// Mitsubishi GX Works2 project: ZhaoQing_HuaCheng1_12_15_8_55   PLC: Q03UDE

TYPE ConveyorIO : STRUCT
  xCWPresent : BOOL;  (* 正转检测有无传感器 *)
  xCCWPresent : BOOL;  (* 反转检测有无传感器 *)
  xLoad : BOOL;  (* 上料请求 *)
  xUnload : BOOL;  (* 下料请求 *)
  xMotorCW : BOOL;  (* 电机正转 *)
  xMotorCCW : BOOL;  (* 电机反转 *)
  xEmpty : BOOL;  (* 线体状态为空 *)
  xNextRun : BOOL;  (* 下段线体运行 *)
  xUnloadCCW : BOOL;  (* 下料为反转 *)
  xloadCCW : BOOL;  (* 上料为反转 *)
  xForward : BOOL;  (* 正转手动 *)
  xBackward : BOOL;  (* 反转手动 *)
  xBusy : BOOL;  (* 工作中 *)
  xPutInto : BOOL;  (* 线体直接投入物料 *)
  xLoadAlarrm : BOOL;  (* 上料报警 *)
  xUnloadAlarm : BOOL;  (* 下料报警 *)
  iProductCategory : INT;  (* 产品种类 *)
  tLoadDelay : TIME;  (* 进入延时设置 *)
  tUnloadAlarmDelay : TIME;  (* 下料时间设置 *)
  xNotArriveAlarm : BOOL;  (* 未到达报警 *)
END_STRUCT END_TYPE

TYPE ShuttleCarIO : STRUCT
  xReady : BOOL;  (* 准备就绪 *)
  xForward : BOOL;  (* 正转 *)
  xBackward : BOOL;  (* 反转 *)
  iCurrentPos : INT;  (* 当前位置 *)
  iDestinationPos : INT;  (* 目标位置 *)
  xCW : BOOL;  (* 正转输出 *)
  xCCW : BOOL;  (* 反转输出 *)
  xBrake : BOOL;  (* 刹车 *)
  xHomeSwitch : BOOL;  (* 零位接近开关 *)
  xPosLimit : BOOL;  (* 正限位 *)
  xNegLimit : BOOL;  (* 负限位 *)
  xMDIExe : BOOL;  (* MDI开始 *)
  xMDIDone : BOOL;  (* MDI 完成 *)
  xPassLimit : BOOL;  (* 限位屏蔽 *)
  xPosLimitCatch : BOOL;  (* 正限位捕捉 *)
  xNegLimitCatch : BOOL;  (* 负限位捕捉 *)
  xHomeExe : BOOL;  (* 开始寻零 *)
  xHomeDone : BOOL;  (* 寻零完成 *)
  xHomeBusy : BOOL;  (* 寻零中 *)
  xHomeFailed : BOOL;  (* 寻零失败 *)
  xBusy : BOOL;  (* 工作中 *)
END_STRUCT END_TYPE

TYPE SwitchIO : STRUCT
  xLiftCylinderRetractDetect : BOOL;
  xLiftCylinderExtendDetect : BOOL;
  xLiftCylinderRetract : BOOL;
  xLiftCylinderExtend : BOOL;
  xEntryBarCylinderRetract : BOOL;
  xLiftCylinderExtendInit : BOOL;
  xEntryEnable : BOOL;
  xExitEnable : BOOL;
  xExitBarCylinderRetract : BOOL;
  xSwithEnable : BOOL;
  xLiftCylinderRetractButton : BOOL;
  xLiftCylinderExtendButton : BOOL;
  xEntryBarCylinderRetractButton : BOOL;
  xExitBarCylinderRetractButton : BOOL;
END_STRUCT END_TYPE

// global labels: Global1
VAR_GLOBAL
  g_xAuto : BOOL;
  g_xManual : BOOL;
  g_xEStop AT X23 : BOOL;
  g_xReset AT X20 : BOOL;
  g_xStackLampRed AT Y120 : BOOL;
  g_xStackLampAmber AT Y121 : BOOL;
  g_xStackLampGreen AT Y122 : BOOL;
  g_xBuzzer AT Y123 : BOOL;
  g_xStop AT M2 : BOOL;
  g_xLocalAutoStart AT M1 : BOOL;
  g_xRemoteAutoStart AT M0 : BOOL;
  g_xRemoteAuto AT M10 : BOOL;
  g_iState AT D40 : INT;
  g_iLocalAutoStep : INT;
  g_xAlarm : BOOL;
END_VAR

// task Task_01 (event TRUE, interval 0, priority 31): POU, Start, UDP

PROGRAM POU
VAR
  H3000Conveyor1 : Conveyor;
  H3000Conveyor1IO : ConveyorIO;
  H3000Conveyor2 : Conveyor;
  H3000Conveyor2IO : ConveyorIO;
  H3000Conveyor3 : Conveyor;
  H3000Conveyor3IO : ConveyorIO;
  H3000Conveyor4 : Conveyor;
  H3000Conveyor4IO : ConveyorIO;
  H3000Conveyor5 : Conveyor;
  H3000Conveyor5IO : ConveyorIO;
  H3000Conveyor6 : Conveyor;
  H3000Conveyor6IO : ConveyorIO;
  H3000Conveyor7 : Conveyor;
  H3000Conveyor7IO : ConveyorIO;
  H3000Conveyor8 : Conveyor;
  H3000Conveyor8IO : ConveyorIO;
  H3000Conveyor9 : Conveyor;
  H3000Conveyor9IO : ConveyorIO;
  H3000Conveyor10 : Conveyor;
  H3000Conveyor10IO : ConveyorIO;
  H3000ChemConveyor1 : Conveyor;
  H3000ChemConveyor1IO : ConveyorIO;
  H3000ChemConveyor2 : Conveyor;
  H3000ChemConveyor2IO : ConveyorIO;
  H3000ChemConveyor3 : Conveyor;
  H3000ChemConveyor3IO : ConveyorIO;
  Lifter1 : ShuttleCar;
  Lifter1IO : ShuttleCarIO;
  Conveyor1 : Conveyor;
  Conveyor1IO : ConveyorIO;
  Lifter2 : ShuttleCar;
  Lifter2IO : ShuttleCarIO;
  Conveyor2 : Conveyor;
  Conveyor2IO : ConveyorIO;
  H2200Conveyor1 : Conveyor;
  H2200Conveyor1IO : ConveyorIO;
  H2200Conveyor2 : Conveyor;
  H2200Conveyor2IO : ConveyorIO;
  H2200Conveyor3 : Conveyor;
  H2200Conveyor3IO : ConveyorIO;
  H2200Conveyor4 : Conveyor;
  H2200Conveyor4IO : ConveyorIO;
  H2200Conveyor5 : Conveyor;
  H2200Conveyor5IO : ConveyorIO;
  H2200Conveyor6 : Conveyor;
  H2200Conveyor6IO : ConveyorIO;
  H2200Conveyor7 : Conveyor;
  H2200Conveyor7IO : ConveyorIO;
  H2200Conveyor8 : Conveyor;
  H2200Conveyor8IO : ConveyorIO;
  H2200Conveyor9 : Conveyor;
  H2200Conveyor9IO : ConveyorIO;
  H2200Conveyor10 : Conveyor;
  H2200Conveyor10IO : ConveyorIO;
  H1000Conveyor1 : Conveyor;
  H1000Conveyor1IO : ConveyorIO;
  H1000Conveyor2 : Conveyor;
  H1000Conveyor2IO : ConveyorIO;
  H1000Conveyor3 : Conveyor;
  H1000Conveyor3IO : ConveyorIO;
  H1000Conveyor4 : Conveyor;
  H1000Conveyor4IO : ConveyorIO;
  H1000Conveyor5 : Conveyor;
  H1000Conveyor5IO : ConveyorIO;
  H1000Conveyor6 : Conveyor;
  H1000Conveyor6IO : ConveyorIO;
  H1000Conveyor7 : Conveyor;
  H1000Conveyor7IO : ConveyorIO;
  H1000Conveyor8 : Conveyor;
  H1000Conveyor8IO : ConveyorIO;
  H1000Conveyor9 : Conveyor;
  H1000Conveyor9IO : ConveyorIO;
  H3000SwitchChem : Switch;
  H3000SwitchChemIO : SwitchIO;
  H850Switch : Switch;
  H850SwitchIO : SwitchIO;
  H850SwitchConveyorIn : ConveyorIO;
  H850SwitchConveyorOut : ConveyorIO;
  H850Conveyor8 : Conveyor;
  H850Conveyor8IO : ConveyorIO;
  H1000Conveyor10 : Conveyor;
  H1000Conveyor10IO : ConveyorIO;
  H3000SwitchChemConveyorIn : ConveyorIO;
  H3000SwitchChemConveyorOut : ConveyorIO;
  H3000SwitchQuadPackage : Switch;
  H3000SwitchQuadPackageIO : SwitchIO;
  H3000SwitchPackageConveyorIn : ConveyorIO;
  H3000SwitchPackageConveyorOut : ConveyorIO;
  H2200Switch1 : Switch;
  H2200Switch1IO : SwitchIO;
  H2200Switch1ConveyorIn : ConveyorIO;
  H2200Switch1ConveyorOut : ConveyorIO;
  H2200Switch2 : Switch;
  H2200Switch2IO : SwitchIO;
  H2200Switch2ConveyorIn : ConveyorIO;
  H2200Switch2ConveyorOut : ConveyorIO;
  iStep : INT;
  Import1Conveyor1 : Conveyor;
  Import1Conveyor1IO : ConveyorIO;
  Import1Conveyor2 : Conveyor;
  Import1Conveyor2IO : ConveyorIO;
  Import2Conveyor1 : Conveyor;
  Import2Conveyor1IO : ConveyorIO;
  Import2Conveyor2 : Conveyor;
  Import2Conveyor2IO : ConveyorIO;
  Export1Conveyor1 : Conveyor;
  Export1Conveyor1IO : ConveyorIO;
  Export1Conveyor2 : Conveyor;
  Export1Conveyor2IO : ConveyorIO;
  Export2Conveyor1 : Conveyor;
  Export2Conveyor1IO : ConveyorIO;
  Export2Conveyor2 : Conveyor;
  Export2Conveyor2IO : ConveyorIO;
  Export2Switch : Switch;
  Export2SwitchIO : SwitchIO;
  Export2SwitchConveyorIn : ConveyorIO;
  Export2SwitchConveyorOut : ConveyorIO;
  H850Rotor : ShuttleCar;
  H850RotorIO : ShuttleCarIO;
  H850RotorConveyor : Conveyor;
  H850RotorConveyorIO : ConveyorIO;
  H2200RotorIO : ShuttleCarIO;
  H2200RotorConveyor : Conveyor;
  H2200RotorConveyorIO : ConveyorIO;
  H2200Rotor : ShuttleCar;
  H850Conveyor1 : Conveyor;
  H850Conveyor1IO : ConveyorIO;
  H850Conveyor3 : Conveyor;
  H850Conveyor3IO : ConveyorIO;
  H850Conveyor4 : Conveyor;
  H850Conveyor4IO : ConveyorIO;
  H850Conveyor5 : Conveyor;
  H850Conveyor5IO : ConveyorIO;
  H850Conveyor6 : Conveyor;
  H850Conveyor6IO : ConveyorIO;
  Lifter2Position : ARRAY [0..5] OF INT;
  ii : INT;  (* 提升机2任务号 *)
  H2200SwitchEmptyABack : Switch;
  H2200SwitchEmptyABackIO : SwitchIO;
  H2200SwitchEmptyABackConveyorIn : ConveyorIO;
  H2200SwitchEmptyABackConveyorOut : ConveyorIO;
  H2200SwitchEmptyBBack : Switch;
  H2200SwitchEmptyBBackIO : SwitchIO;
  H2200SwitchEmptyBBackConveyorIn : ConveyorIO;
  H2200SwitchEmptyBBackConveyorOut : ConveyorIO;
  H2200ImportConveyor1 : Conveyor;
  H2200ImportConveyor1IO : ConveyorIO;
  H2200ImportConveyor2 : Conveyor;
  H2200ImportConveyor2IO : ConveyorIO;
  Import1Switch : Switch;
  Import1SwitchIO : SwitchIO;
  Import1SwitchConveyorIn : ConveyorIO;
  Import1SwitchConveyorOut : ConveyorIO;
  Export1Switch : Switch;
  Export1SwitchIO : SwitchIO;
  Export1SwitchConveyorIn : ConveyorIO;
  Export1SwitchConveyorOut : ConveyorIO;
  Import2Switch : Switch;
  Import2SwitchIO : SwitchIO;
  Import2SwitchConveyorIn : ConveyorIO;
  Import2SwitchConveyorOut : ConveyorIO;
  Import1LoadCylinder : ShuttleCar;
  Import1LoadCylinderIO : ShuttleCarIO;
  Import2LoadCylinder : ShuttleCar;
  Import2LoadCylinderIO : ShuttleCarIO;
  Export1LoadCylinder : ShuttleCar;
  Export1LoadCylinderIO : ShuttleCarIO;
  Export2LoadCylinder : ShuttleCar;
  Export2LoadCylinderIO : ShuttleCarIO;
  Lifter2ExportChem : BOOL;  (* 提升机2满框去化成 *)
  Lifter2TaskID : INT;  (* 提升机2动作步骤 *)
  Lifter2Task : PriorityFB;
  H2200Switch1Task : PriorityFB;
  H2200Switch1TaskID : INT;
  H2200Switch1EmptyImport : BOOL;  (* 空框返回入库 *)
  Lifter1Speed : ShuttleCarVelocityFB;
END_VAR
H3000SwitchQuadPackage(ConveyorEntryIO:=H3000SwitchPackageConveyorIn ,
                                                        ConveyorExitIO:=H3000SwitchPackageConveyorOut ,
                                                        SwitchIO:=H3000SwitchQuadPackageIO );
H3000SwitchQuadPackageIO.xLiftCylinderExtendButton:=M75;
H3000SwitchQuadPackageIO.xLiftCylinderRetractButton:=M76;
H3000SwitchQuadPackageIO.xExitBarCylinderRetractButton:=M83;
Y128:=H3000SwitchQuadPackageIO.xEXITBarCylinderRetract;
Y12C:=H3000SwitchQuadPackageIO.xLiftCylinderExtend;
Y12A:=H3000SwitchQuadPackageIO.xLiftCylinderRetract;
H3000SwitchQuadPackageIO.xLiftCylinderExtendDetect:=X29;
H3000SwitchQuadPackageIO.xLiftCylinderRetractDetect:=X2A;
H3000SwitchPackageConveyorIn.xForward:=M77;
H3000SwitchPackageConveyorIn.xCWPresent:=X28;
(*Y187:=H3000SwitchPackageConveyorIn.xMotorCW;*)
H3000SwitchPackageConveyorOut.xForward:=M78;
H3000SwitchPackageConveyorOut.xCWPresent:=X2B;
Y12B:=H3000SwitchPackageConveyorOut.xMotorCW;

H3000SwitchChem(ConveyorEntryIO:=H3000SwitchChemConveyorIn ,
                                                        ConveyorExitIO:=H3000SwitchChemConveyorOut ,
                                                        SwitchIO:=H3000SwitchChemIO );
H3000SwitchChemIO.xLiftCylinderExtendButton:=M79;
H3000SwitchChemIO.xLiftCylinderRetractButton:=M80;
Y129:=H3000SwitchChemIO.xLiftCylinderExtend;
Y12D:=H3000SwitchChemIO.xLiftCylinderRetract;
H3000SwitchChemIO.xLiftCylinderExtendDetect:=X2C;
H3000SwitchChemIO.xLiftCylinderRetractDetect:=X2D;
H3000SwitchChemConveyorIn.xForward:=M81;
H3000SwitchChemConveyorIn.xCWPresent:=X27;
(*Y19B:=H3000SwitchPackageConveyorIn.xMotorCW;*)
H3000SwitchChemConveyorOut.xForward:=M82;
H3000SwitchChemConveyorOut.xCWPresent:=X2E;
Y12E:=H3000SwitchChemConveyorOut.xMotorCW;
H3000SwitchChemIO.xSwithEnable:=1;

Lifter1(ShuttleCarInOut:=Lifter1IO);
ShuttleCarCurrentPosition(X8C OR X8D ,X8C ,X8D, FALSE, Lifter1IO.iCurrentPos);
Lifter1Speed(xEnable:= g_xAuto,
                        xMotorCW:= Lifter1IO.xCW ,
                        xMotorCCW:= Lifter1IO.xCCW,
                        xPosition1Switch:= X8C,
                        xDecelerationSwitch:= X8B ,
	                    xPosition2Switch:= X8D ,
	                    xHighSpeed:= Y18F );
Lifter1IO.xReady:=X24;
Lifter1Io.xForward:=M50 OR X91;
Lifter1IO.xBackward:=M51 OR X92;
Lifter1IO.xPosLimit:=X8E;
Lifter1IO.xNegLimit:=X8F;
Y18D:=Lifter1IO.xCW;
Y18E:=Lifter1IO.xCCW;
Y192:=Lifter1IO.xBrake;

Conveyor1(ConveyorMotor:=Conveyor1IO);
Conveyor1IO.xForward:=M52;
Conveyor1IO.xBackward:=M53;
Conveyor1IO.xCWPresent:=X93;
Conveyor1IO.xCCWPresent:=X94;
Y18B:=Conveyor1IO.xMotorCW;
Y18C:=Conveyor1IO.xMotorCCW;
(*2号提升机*)
Lifter2(ShuttleCarInOut:=Lifter2IO);
Lifter2Position[0]:=0;
Lifter2Position[1]:=57;
Lifter2Position[2]:=590;
Lifter2Position[3]:=5828;
Lifter2Position[4]:=6202;
Lifter2Position[5]:=9200;
Y195:=ShuttleCarVelocityEncoder( g_xAuto , D190 , Lifter2Position[Lifter2IO.iDestinationPos] );
IF LDP(TRUE,g_xAuto) THEN
	Lifter2IO.iCurrentPos:=0;
END_IF;
FOR ii:=0 TO 5 BY 1 DO
	IF abs(D190-Lifter2Position[ii])<5 THEN
		Lifter2IO.iCurrentPos:=ii;
	END_IF;
END_FOR;
Lifter2IO.xReady:=X25;
(*提升机占用标志位控制*)
Lifter2Task(xCondition1:= NOT H850Conveyor8IO.xEmpty ,
                     xCondition2:= NOT H1000Conveyor1IO.xEmpty ,
                     xCondition3:= NOT H3000ChemConveyor3IO.xEmpty  AND Lifter2ExportChem ,
                     xCondition4:= NOT H3000ChemConveyor3IO.xEmpty  AND NOT Lifter2ExportChem ,
                     xCondition5:= FALSE ,
	                 xTaskComplete:= (Lifter2IO.iCurrentPos=3 OR Lifter2IO.iCurrentPos=4) AND LDP(TRUE,Conveyor2IO.xEmpty)  ,
	                 xReset:= g_xReset,
	                 iPriority:=  Lifter2TaskID );
Lifter2Io.xForward:=M54 OR X9B;
Lifter2IO.xBackward:=M55 OR X9C;
Lifter2IO.xPosLimit:=X98;
Lifter2IO.xNegLimit:=X99;
Y193:=Lifter2IO.xCW;
Y194:=Lifter2IO.xCCW;
Y198:=Lifter2IO.xBrake;
(*提升机2编码器清零，到达负限位后清零*)
IF NOT Lifter2IO.xNegLimit THEN
	Y125:=1;
ELSE
	Y125:=0;
END_IF;

Conveyor2(ConveyorMotor:=Conveyor2IO);
Conveyor2IO.xForward:=M56;
Conveyor2IO.xBackward:=M57;
Conveyor2IO.xCWPresent:=X9D;
Conveyor2IO.xCCWPresent:=X9E;
Y19A:=Conveyor2IO.xMotorCW;
Y199:=Conveyor2IO.xMotorCCW;

(*去二封线体*)
H3000Conveyor1(ConveyorMotor:=H3000Conveyor1IO);
H3000Conveyor1IO.xForward:=M30;
H3000Conveyor1IO.xCWPresent:=X2F;
Y12F:=H3000Conveyor1IO.xMotorCW;

H3000Conveyor2(ConveyorMotor:=H3000Conveyor2IO);
H3000Conveyor2IO.xForward:=M31;
H3000Conveyor2IO.xCWPresent:=X30;
Y130:=H3000Conveyor2IO.xMotorCW;

H3000Conveyor3(ConveyorMotor:=H3000Conveyor3IO);
H3000Conveyor3IO.xForward:=M32;
H3000Conveyor3IO.xCWPresent:=X31;
Y131:=H3000Conveyor3IO.xMotorCW;

H3000Conveyor4(ConveyorMotor:=H3000Conveyor4IO);
H3000Conveyor4IO.xForward:=M33;
H3000Conveyor4IO.xCWPresent:=X32;
Y132:=H3000Conveyor4IO.xMotorCW;

H3000Conveyor5(ConveyorMotor:=H3000Conveyor5IO);
H3000Conveyor5IO.xForward:=M34;
H3000Conveyor5IO.xCWPresent:=X33;
Y133:=H3000Conveyor5IO.xMotorCW;

H3000Conveyor6(ConveyorMotor:=H3000Conveyor6IO);
H3000Conveyor6IO.xForward:=M34;
H3000Conveyor6IO.xCWPresent:=X34;
Y134:=H3000Conveyor6IO.xMotorCW;

H3000Conveyor7(ConveyorMotor:=H3000Conveyor7IO);
H3000Conveyor7IO.xForward:=M35;
H3000Conveyor7IO.xCWPresent:=X35;
Y135:=H3000Conveyor7IO.xMotorCW;
H3000Conveyor8(ConveyorMotor:=H3000Conveyor8IO);
H3000Conveyor8IO.xForward:=M36;
H3000Conveyor8IO.xCWPresent:=X36;
Y136:=H3000Conveyor8IO.xMotorCW;

H3000Conveyor9(ConveyorMotor:=H3000Conveyor9IO);
H3000Conveyor9IO.xForward:=M37;
H3000Conveyor9IO.xCWPresent:=X37;
Y137:=H3000Conveyor9IO.xMotorCW;

H3000Conveyor10(ConveyorMotor:=H3000Conveyor10IO);
H3000Conveyor10IO.xForward:=M38;
H3000Conveyor10IO.xCWPresent:=X38;
Y138:=H3000Conveyor10IO.xMotorCW;

(*本段线体没有接线*)
(*H3000ChemConveyor1(ConveyorMotor:=H3000ChemConveyor1IO);
H3000ChemConveyor1IO.xForward:=M39;
H3000ChemConveyor1IO.xCWPresent:=X39;
Y139:=H3000ChemConveyor1IO.xMotorCW;*)

(*去化成H3000线体*)
H3000ChemConveyor2(ConveyorMotor:=H3000ChemConveyor2IO);
H3000ChemConveyor2IO.xForward:=M40;
H3000ChemConveyor2IO.xCWPresent:=X39;
Y13A:=H3000ChemConveyor2IO.xMotorCW;

H3000ChemConveyor3(ConveyorMotor:=H3000ChemConveyor3IO);
H3000ChemConveyor3IO.xForward:=M41;
H3000ChemConveyor3IO.xCWPresent:=X3B;
Y13B:=H3000ChemConveyor3IO.xMotorCW;
(*入库线体*)
H2200Switch1(ConveyorEntryIO:=H2200Switch1ConveyorIn ,
                                                        ConveyorExitIO:=H2200Switch1ConveyorOut ,
                                                        SwitchIO:=H2200Switch1IO );
H2200Switch1Task(xCondition1:=NOT  H2200SwitchEmptyABackConveyorIn.xEmpty AND H2200Switch1EmptyImport,
                                    xCondition2:= NOT  H2200SwitchEmptyBBackConveyorIn.xEmpty AND H2200Switch1EmptyImport,
                                    xCondition3:=NOT  H2200SwitchEmptyABackConveyorIn.xEmpty AND NOT H2200Switch1EmptyImport  ,
                                    xCondition4:=(* NOT  H2200SwitchEmptyBBackConveyorIn.xEmpty AND NOT H2200Switch1EmptyImport*)FALSE,
                                    xCondition5:= NOT H2200ImportConveyor2IO.xEmpty  ,
	                               xTaskComplete:= LDP(TRUE, H2200Switch1ConveyorIn.xEmpty) OR LDP(TRUE, H2200Switch1ConveyorOut.xEmpty)  ,
	                               xReset:= g_xReset ,
	                               iPriority:= H2200Switch1TaskID);
H2200Switch1IO.xLiftCylinderExtendButton:=M84;
H2200Switch1IO.xLiftCylinderRetractButton:=M85;
H2200Switch1IO.xExitBarCylinderRetractButton:=M86;
Y158:=H2200Switch1IO.xEXITBarCylinderRetract;
Y155:=H2200Switch1IO.xLiftCylinderExtend;
Y156:=H2200Switch1IO.xLiftCylinderRetract;
H2200Switch1IO.xLiftCylinderExtendDetect:=X55;
H2200Switch1IO.xLiftCylinderRetractDetect:=X56;
H2200Switch1ConveyorIn.xForward:=M87;
H2200Switch1ConveyorIn.xCWPresent:=X57;
(*Y177:=H2200Switch1ConveyorIn.xMotorCW;*)
H2200Switch1ConveyorOut .xForward:=M88;
H2200Switch1ConveyorOut .xCWPresent:=X57;
H2200Switch1ConveyorOut.tLoadDelay:=T#1s;
Y157:=H2200Switch1ConveyorOut .xMotorCW;

H2200ImportConveyor1(ConveyorMotor:=H2200ImportConveyor1IO);
H2200ImportConveyor1IO.xForward:=M136;
H2200ImportConveyor1IO.xCWPresent:=X53;
Y153:=H2200ImportConveyor1IO.xMotorCW;

H2200ImportConveyor2(ConveyorMotor:=H2200ImportConveyor2IO);
H2200ImportConveyor2IO.xForward:=M122;
H2200ImportConveyor2IO.xCWPresent:=X58;
Y154:=H2200ImportConveyor2IO.xMotorCW;


H2200Switch2(ConveyorEntryIO:=H2200Switch2ConveyorIn ,
                                                        ConveyorExitIO:=H2200Switch2ConveyorOut ,
                                                        SwitchIO:=H2200Switch2IO );
H2200Switch2IO.xLiftCylinderExtendButton:=M89;
H2200Switch2IO.xLiftCylinderRetractButton:=M90;
H2200Switch2IO.xExitBarCylinderRetractButton:=M91;
Y15C:=H2200Switch2IO.xEXITBarCylinderRetract;
Y159:=H2200Switch2IO.xLiftCylinderExtend;
Y15A:=H2200Switch2IO.xLiftCylinderRetract;
H2200Switch2IO.xLiftCylinderExtendDetect:=X59;
H2200Switch2IO.xLiftCylinderRetractDetect:=X5A;
H2200Switch2ConveyorIn.xForward:=M92;
H2200Switch2ConveyorIn.xCWPresent:=X5B;
H2200Switch2ConveyorIn.tLoadDelay:=T#4s;
Y15B:=H2200Switch2ConveyorIn.xMotorCW;
H2200Switch2ConveyorOut .xForward:=M93;
H2200Switch2ConveyorOut .xCWPresent:=X5B;
Y186:=H2200Switch2ConveyorOut.xMotorCW;(*	Y186:=1;(***入库倍速链***)
H2200Switch2IO.xLiftCylinderExtendInit:=1;

H2200SwitchEmptyABack(ConveyorEntryIO:=H2200SwitchEmptyABackConveyorIn ,
                                                        ConveyorExitIO:=H2200SwitchEmptyABackConveyorOut ,
                                                        SwitchIO:=H2200SwitchEmptyABackIO );
H2200SwitchEmptyABackIO.xLiftCylinderExtendButton:=M137;
H2200SwitchEmptyABackIO.xLiftCylinderRetractButton:=M138;
H2200SwitchEmptyABackIO.xExitBarCylinderRetractButton:=M139;
Y160:=H2200SwitchEmptyABackIO.xLiftCylinderExtend;
Y161:=H2200SwitchEmptyABackIO.xLiftCylinderRetract;
H2200SwitchEmptyABackIO.xLiftCylinderExtendDetect:=X60;
H2200SwitchEmptyABackIO.xLiftCylinderRetractDetect:=X61;
H2200SwitchEmptyABackConveyorIn.xForward:=M140;
H2200SwitchEmptyABackConveyorIn.xCWPresent:=X62;
H2200SwitchEmptyABackConveyorIn.tLoadDelay:=T#2s;
Y162:=H2200SwitchEmptyABackConveyorIn.xMotorCW;
H2200SwitchEmptyABackConveyorOut .xForward:=M146;
H2200SwitchEmptyABackConveyorOut.xCWPresent:=X62;
(*空框返回共同倍速链*)
Y177:=H2200SwitchEmptyABackConveyorOut .xMotorCW OR H2200SwitchEmptyBBackConveyorOut .xMotorCW ;

(*H2200SwitchEmptyBBack(ConveyorEntryIO:=H2200SwitchEmptyBBackConveyorIn ,
                                                        ConveyorExitIO:=H2200SwitchEmptyBBackConveyorOut ,
                                                        SwitchIO:=H2200SwitchEmptyBBackIO );
H2200SwitchEmptyBBackIO.xLiftCylinderExtendButton:=M141;
H2200SwitchEmptyBBackIO.xLiftCylinderRetractButton:=M142;
H2200SwitchEmptyBBackIO.xExitBarCylinderRetractButton:=M143;
Y166:=H2200SwitchEmptyBBackIO.xLiftCylinderExtend;
Y167:=H2200SwitchEmptyBBackIO.xLiftCylinderRetract;
H2200SwitchEmptyBBackIO.xLiftCylinderExtendDetect:=X66;
H2200SwitchEmptyBBackIO.xLiftCylinderRetractDetect:=X67;
H2200SwitchEmptyBBackConveyorIn.xForward:=M144;
H2200SwitchEmptyBBackConveyorIn.xCWPresent:=X68;
H2200SwitchEmptyBBackConveyorIn.tLoadDelay:=T#2s;
Y168:=H2200SwitchEmptyBBackConveyorIn.xMotorCW;
H2200SwitchEmptyBBackConveyorOut .xForward:=M145;
H2200SwitchEmptyBBackConveyorOut.xCWPresent:=X68;
H2200SwitchEmptyBBackConveyorOut.tLeaveDelay:=T#30S;*)
(*空框回注液转台*)
H2200Rotor(ShuttleCarInOut:=H2200RotorIO);
ShuttleCarCurrentPosition(X6F OR X75 ,X6F ,X75, FALSE,H2200RotorIO.iCurrentPos );
H2200RotorIO.xReady:=TRUE;
H2200RotorIO.xForward:=M78;
H2200RotorIO.xBackward:=M79;
H2200RotorIO.xPosLimit:=X71;
H2200RotorIO.xNegLimit:=X72;
Y170:=H2200RotorIO.xCW;
Y16F:=H2200RotorIO.xCCW;
Y1B8:=H2200RotorIO.xBrake;

H2200RotorConveyor(ConveyorMotor:=H2200RotorConveyorIO);
H2200RotorConveyorIO.xForward:=M80;
H2200RotorConveyorIO.xBackward:=M81;
H2200RotorConveyorIO.xCWPresent:=X74;
H2200RotorConveyorIO.xCcWPresent:=X73;
Y172:=H2200RotorConveyorIO.xMotorCW;
Y171:=H2200RotorConveyorIO.xMotorCCW;
(*去化成H2200线体*)
H2200Conveyor1(ConveyorMotor:=H2200Conveyor1IO);
H2200Conveyor1IO.xForward:=M42;
H2200Conveyor1IO.xCWPresent:=X3F;
Y13F:=H2200Conveyor1IO.xMotorCW;

H2200Conveyor2(ConveyorMotor:=H2200Conveyor2IO);
H2200Conveyor2IO.xForward:=M43;
H2200Conveyor2IO.xCWPresent:=X40;
Y140:=H2200Conveyor2IO.xMotorCW;

H2200Conveyor3(ConveyorMotor:=H2200Conveyor3IO);
H2200Conveyor3IO.xForward:=M44;
H2200Conveyor3IO.xCWPresent:=X41;
Y141:=H2200Conveyor3IO.xMotorCW;

(*H2200Conveyor4(ConveyorMotor:=H2200Conveyor4IO);
H2200Conveyor4IO.xForward:=M45;
H2200Conveyor4IO.xCWPresent:=X42;
Y142:=H2200Conveyor4IO.xMotorCW;

H2200Conveyor5(ConveyorMotor:=H2200Conveyor5IO);
H2200Conveyor5IO.xForward:=M46;
H2200Conveyor5IO.xCWPresent:=X43;
Y143:=H2200Conveyor5IO.xMotorCW;

H2200Conveyor6(ConveyorMotor:=H2200Conveyor6IO);
H2200Conveyor6IO.xForward:=M47;
H2200Conveyor6IO.xCWPresent:=X44;
Y144:=H2200Conveyor6IO.xMotorCW;

H2200Conveyor7(ConveyorMotor:=H2200Conveyor7IO);
H2200Conveyor7IO.xForward:=M48;
H2200Conveyor7IO.xCWPresent:=X45;
Y145:=H2200Conveyor7IO.xMotorCW;

H2200Conveyor8(ConveyorMotor:=H2200Conveyor8IO);
H2200Conveyor8IO.xForward:=M49;
H2200Conveyor8IO.xCWPresent:=X46;
Y146:=H2200Conveyor8IO.xMotorCW;

H2200Conveyor9(ConveyorMotor:=H2200Conveyor9IO);
H2200Conveyor9IO.xForward:=M58;
H2200Conveyor9IO.xCWPresent:=X47;
Y147:=H2200Conveyor9IO.xMotorCW;

H2200Conveyor10(ConveyorMotor:=H2200Conveyor10IO);
H2200Conveyor10IO.xForward:=M59;
H2200Conveyor10IO.xCWPresent:=X48;
Y148:=H2200Conveyor10IO.xMotorCW;
(*去化成回流H1100线体*)
H1000Conveyor1(ConveyorMotor:=H1000Conveyor1IO);
H1000Conveyor1IO.xForward:=M60;
H1000Conveyor1IO.xCWPresent:=X49;
Y149:=H1000Conveyor1IO.xMotorCW;

(*H1000Conveyor2(ConveyorMotor:=H1000Conveyor2IO);
H1000Conveyor2IO.xForward:=M61;
H1000Conveyor2IO.xCWPresent:=X4A;
Y14A:=H1000Conveyor2IO.xMotorCW;

H1000Conveyor3(ConveyorMotor:=H1000Conveyor3IO);
H1000Conveyor3IO.xForward:=M62;
H1000Conveyor3IO.xCWPresent:=X4B;
Y14B:=H1000Conveyor3IO.xMotorCW;

H1000Conveyor4(ConveyorMotor:=H1000Conveyor4IO);
H1000Conveyor4IO.xForward:=M63;
H1000Conveyor4IO.xCWPresent:=X4C;
Y14C:=H1000Conveyor4IO.xMotorCW;

H1000Conveyor5(ConveyorMotor:=H1000Conveyor5IO);
H1000Conveyor5IO.xForward:=M64;
H1000Conveyor5IO.xCWPresent:=X4D;
Y14D:=H1000Conveyor5IO.xMotorCW;

H1000Conveyor6(ConveyorMotor:=H1000Conveyor6IO);
H1000Conveyor6IO.xForward:=M65;
H1000Conveyor6IO.xCWPresent:=X4E;
Y14E:=H1000Conveyor6IO.xMotorCW;

H1000Conveyor7(ConveyorMotor:=H1000Conveyor7IO);
H1000Conveyor7IO.xForward:=M66;
H1000Conveyor7IO.xCWPresent:=X4F;
Y14F:=H1000Conveyor7IO.xMotorCW;

H1000Conveyor8(ConveyorMotor:=H1000Conveyor8IO);
H1000Conveyor8IO.xForward:=M67;
H1000Conveyor8IO.xCWPresent:=X50;
Y150:=H1000Conveyor8IO.xMotorCW;

H1000Conveyor9(ConveyorMotor:=H1000Conveyor9IO);
H1000Conveyor9IO.xForward:=M68;
H1000Conveyor9IO.xCWPresent:=X51;
Y151:=H1000Conveyor9IO.xMotorCW;*)

H1000Conveyor10(ConveyorMotor:=H1000Conveyor10IO);
H1000Conveyor10IO.xForward:=M67;
H1000Conveyor10IO.xCWPresent:=X52;
Y152:=H1000Conveyor10IO.xMotorCW;

(*注液入与出线体*)
H850Conveyor1(ConveyorMotor:=H850Conveyor1IO);
H850Conveyor1IO.xForward:=M129;
H850Conveyor1IO.xCWPresent:=X78;
Y178:=H850Conveyor1IO.xMotorCW;

H850Conveyor3(ConveyorMotor:=H850Conveyor3IO);
H850Conveyor3IO.xForward:=M130;
H850Conveyor3IO.xCWPresent:=X7A;
Y17A:=H850Conveyor3IO.xMotorCW;

H850Conveyor4(ConveyorMotor:=H850Conveyor4IO);
H850Conveyor4IO.xForward:=M131;
H850Conveyor4IO.xCWPresent:=X7B;
Y17B:=H850Conveyor4IO.xMotorCW;

H850Conveyor5(ConveyorMotor:=H850Conveyor5IO);
H850Conveyor5IO.xForward:=M132;
H850Conveyor5IO.xCWPresent:=X7C;
Y17C:=H850Conveyor5IO.xMotorCW;

H850Conveyor6(ConveyorMotor:=H850Conveyor6IO);
H850Conveyor6IO.xForward:=M133;
H850Conveyor6IO.xCWPresent:=X7D;
Y17D:=H850Conveyor6IO.xMotorCW;

H850Rotor(ShuttleCarInOut:=H850RotorIO);
ShuttleCarCurrentPosition(X82 OR X76  ,X82 ,X76, FALSE,H850RotorIO.iCurrentPos);
H850RotorIO.xReady:=TRUE;
H850RotorIO.xForward:=M75;
H850RotorIO.xBackward:=M76;
H850RotorIO.xPosLimit:=X84;
H850RotorIO.xNegLimit:=X85;
Y182:=H850RotorIO.xCW;
Y183:=H850RotorIO.xCCW;
Y1B9:=H850RotorIO.xBrake;

H850RotorConveyor(ConveyorMotor:=H850RotorConveyorIO);
H850RotorConveyorIO.xForward:=M77;
H850RotorConveyorIO.xBackward:=M82;
H850RotorConveyorIO.xCWPresent:=X87;
H850RotorConveyorIO.xCCWPresent:=X86;
Y185:=H850RotorConveyorIO.xMotorCW;
Y184:=H850RotorConveyorIO.xMotorCCW;
H850RotorConveyorIO.xUnloadCCW:=1;

H850Switch(ConveyorEntryIO:=H850SwitchConveyorIn,ConveyorExitIO:=H850SwitchConveyorOut,SwitchIO:=H850SwitchIO);
H850SwitchIO.xLiftCylinderExtendButton:=M71;
H850SwitchIO.xLiftCylinderRetractButton:=M72;
Y189:=H850SwitchIO.xLiftCylinderExtend;
Y188:=H850SwitchIO.xLiftCylinderRetract;
H850SwitchIO.xLiftCylinderExtendDetect:=X88;
H850SwitchIO.xLiftCylinderRetractDetect:=X89;
H850SwitchConveyorIn.xForward:=M70;
H850SwitchConveyorIn.xCWPresent:=XB4;
Y19B:=H850SwitchConveyorIn.xMotorCW;
H850SwitchConveyorOut.xForward:=M73;
H850SwitchConveyorOut.xCWPresent:=X8A;
Y18A:=H850SwitchConveyorOut.xMotorCW;


H850Conveyor8(ConveyorMotor:=H850Conveyor8IO);
H850Conveyor8IO.xForward:=M74;
H850Conveyor8IO.xCWPresent:=X7F;
Y17F:=H850Conveyor8IO.xMotorCW;

(*高温库前线体*)
(*1巷道入库*)
Import1Conveyor1(ConveyorMotor:=Import1Conveyor1IO);
Import1Conveyor1IO.xForward:=M98;
Import1Conveyor1IO.xCWPresent:=XE3;
Y1F4:=Import1Conveyor1IO.xMotorCW;

Import1Conveyor2(ConveyorMotor:=Import1Conveyor2IO);
Import1Conveyor2IO.tLoadDelay:=T#1s;
Import1Conveyor2IO.xForward:=M99;
Import1Conveyor2IO.xCWPresent:=XE4;
Y1F5:=Import1Conveyor2IO.xMotorCW;

Import1Switch(ConveyorEntryIO:=Import1SwitchConveyorIn,
                          ConveyorExitIO:=Import1SwitchConveyorOut ,
                           SwitchIO:=Import1SwitchIO);
Import1SwitchIO.xLiftCylinderExtendButton:=M147;
Import1SwitchIO.xLiftCylinderRetractButton:=M148;
Import1SwitchIO.xExitBarCylinderRetractButton:=M161;
Y1E0:=Import1SwitchIO.xExitBarCylinderRetract;
Y1E2:=Import1SwitchIO.xLiftCylinderExtend;
Y1E1:=Import1SwitchIO.xLiftCylinderRetract;
Import1SwitchIO.xLiftCylinderExtendDetect:=XE1;
Import1SwitchIO.xLiftCylinderRetractDetect:=XE2;
Import1SwitchConveyorIn.xCWPresent:=XE0;
Import1SwitchConveyorIn.tLoadDelay:=T#2s;
Import1SwitchConveyorOut.xForward:=M149;
Import1SwitchConveyorOut.xCWPresent:=X108;
Y1F6:=Import1SwitchConveyorOut.xMotorCW;

Import1LoadCylinder(ShuttleCarInOut:=Import1LoadCylinderIO);
ShuttleCarCurrentPosition(XE7 OR XE6,XE7 ,XE6, FALSE,Import1LoadCylinderIO.iCurrentPos );
Import1LoadCylinderIO.xReady:=TRUE;
Import1LoadCylinderIO.xForward:=M159;
Import1LoadCylinderIO.xBackward:=M160;
Import1LoadCylinderIO.xPosLimit:=TRUE;
Import1LoadCylinderIO.xNegLimit:=TRUE;
Y1E4:=Import1LoadCylinderIO.xCW;
Y1E3:=Import1LoadCylinderIO.xCCW;

(*1巷道出库*)
Export1Conveyor1(ConveyorMotor:=Export1Conveyor1IO);
Export1Conveyor1IO.xForward:=M94;
Export1Conveyor1IO.xCWPresent:=XEC;
Y1F7:=Export1Conveyor1IO.xMotorCW;

Export1Conveyor2(ConveyorMotor:=Export1Conveyor2iO);
Export1Conveyor2IO.xForward:=M95;
Export1Conveyor2IO.xCWPresent:=XEB;
Y1F8:=Export1Conveyor2IO.xMotorCW;

Export1Switch(ConveyorEntryIO:=Export1SwitchConveyorIn,
                          ConveyorExitIO:=Export1SwitchConveyorOut ,
                           SwitchIO:=Export1SwitchIO);
Export1SwitchIO.xLiftCylinderExtendButton:=M150;
Export1SwitchIO.xLiftCylinderRetractButton:=M151;
Y1E7:=Export1SwitchIO.xLiftCylinderExtend;
Y1E6:=Export1SwitchIO.xLiftCylinderRetract;
Export1SwitchIO.xLiftCylinderExtendDetect:=XE9;
Export1SwitchIO.xLiftCylinderRetractDetect:=XEA;
Export1SwitchConveyorIn.xForward:=M152;
Export1SwitchConveyorIn.xCWPresent:=X106;
Export1SwitchConveyorIn.tLoadDelay:=T#2s;
Y1F9:=Export1SwitchConveyorIn.xMotorCW;
Export1SwitchConveyorOut.xCWPresent:=X106;

Export1LoadCylinder(ShuttleCarInOut:=Export1LoadCylinderIO);
ShuttleCarCurrentPosition(XEF OR XEE ,XEF ,XEE, FALSE,Export1LoadCylinderIO.iCurrentPos);
Export1LoadCylinderIO.xReady:=TRUE;
Export1LoadCylinderIO.xForward:=M157;
Export1LoadCylinderIO.xBackward:=M158;
Export1LoadCylinderIO.xPosLimit:=TRUE;
Export1LoadCylinderIO.xNegLimit:=TRUE;
Y1E9:=Export1LoadCylinderIO.xCW;
Y1E8:=Export1LoadCylinderIO.xCCW;


(*2巷道入库*)
(*Import2Conveyor1(ConveyorMotor:=Import2Conveyor1IO);
Import2Conveyor1IO.xForward:=M153;
Import2Conveyor1IO.xCWPresent:=XF3;
Y1FA:=Import2Conveyor1IO.xMotorCW;

Import2Conveyor2(ConveyorMotor:=Import2Conveyor1IO);
Import2Conveyor2IO.tLoadDelay:=T#1s;
Import2Conveyor2IO.xForward:=M154;
Import2Conveyor2IO.xCWPresent:=XF4;
Y1FB:=Import2Conveyor2IO.xMotorCW;

Import2Switch(ConveyorEntryIO:=Import2SwitchConveyorIn,
                          ConveyorExitIO:=Import2SwitchConveyorOut ,
                           SwitchIO:=Import2SwitchIO);
Import2SwitchIO.xLiftCylinderExtendButton:=M155;
Import2SwitchIO.xLiftCylinderRetractButton:=M156;
Y1ED:=Import2SwitchIO.xLiftCylinderExtend;
Y1EE:=Import2SwitchIO.xLiftCylinderRetract;
Import2SwitchIO.xLiftCylinderExtendDetect:=XF1;
Import2SwitchIO.xLiftCylinderRetractDetect:=XF2;
Import2SwitchConveyorIn.xCWPresent:=X104;
Import2SwitchConveyorIn.tLoadDelay:=T#2s;
Import2SwitchConveyorOut.xForward:=M149;
Import2SwitchConveyorOut.tLeaveDelay:=t#8s;
Import2SwitchConveyorOut.xCWPresent:=XF0;
Y1FC:=Import2SwitchConveyorIn.xMotorCW;

Import2LoadCylinder(ShuttleCarInOut:=Import2LoadCylinderIO);
ShuttleCarCurrentPosition(xf6 or xf7 ,XF6 ,XF7, FALSE,Import2LoadCylinderIO.iCurrentPos );
Import2LoadCylinderIO.xReady:=TRUE;
Import2LoadCylinderIO.xForward:=M161;
Import2LoadCylinderIO.xBackward:=M162;
Import2LoadCylinderIO.xPosLimit:=TRUE;
Import2LoadCylinderIO.xNegLimit:=TRUE;
Y1ED:=Import2LoadCylinderIO.xCW;
Y1EE:=Import2LoadCylinderIO.xCCW;*)

(*2巷道出库*)
(*Export2Conveyor1(ConveyorMotor:=Export2Conveyor1IO);
Export2Conveyor1IO.tLeaveDelay:=t#10s;
Export2Conveyor1IO.xForward:=M96;
Export2Conveyor1IO.xCWPresent:=XFB;
Y1FD:=Export2Conveyor1IO.xMotorCW;

Export2Conveyor2(ConveyorMotor:=Export2Conveyor2iO);
Export2Conveyor2IO.tLeaveDelay:=t#10s;
Export2Conveyor2IO.xForward:=M97;
Export2Conveyor2IO.xCWPresent:=XFC;
Y1FE:=Export2Conveyor2IO.xMotorCW;

Export2Switch(ConveyorEntryIO:=Export2SwitchConveyorIn,
                          ConveyorExitIO:=Export2SwitchConveyorOut ,
                           SwitchIO:=Export2SwitchIO);
Export2SwitchIO.xLiftCylinderExtendButton:=M120;
Export2SwitchIO.xLiftCylinderRetractButton:=M121;
Export2SwitchIO.xLiftCylinderExtendInit:=1;
Y1F1:=Export2SwitchIO.xLiftCylinderExtend;
Y1F0:=Export2SwitchIO.xLiftCylinderRetract;
Export2SwitchIO.xLiftCylinderExtendDetect:=XF9;
Export2SwitchIO.xLiftCylinderRetractDetect:=XFA;
Export2SwitchConveyorIn.xForward:=M123;
Export2SwitchConveyorIn.xCWPresent:=X105;
Y1FF:=Export2SwitchConveyorIn.xMotorCW;
Export2SwitchConveyorOut.xCWPresent:=X105;

(*Export2LoadCylinder(ShuttleCarInOut:=Export2LoadCylinderIO);
ShuttleCarCurrentPosition( XFF OR XFE ,XFF ,XFE, FALSE, Export2LoadCylinderIO.iCurrentPos);
Export2LoadCylinderIO.xReady:=TRUE;
Export2LoadCylinderIO.xForward:=M124;
Export2LoadCylinderIO.xBackward:=M125;
Export2LoadCylinderIO.xPosLimit:=TRUE;
Export2LoadCylinderIO.xNegLimit:=TRUE;
Y1F2:=Export2LoadCylinderIO.xCW;
Y1F3:=Export2LoadCylinderIO.xCCW;*)

IF g_xAuto THEN
	(**高温库前自动程序**)
	Y187:=1;(***出库倍速链***)
	(**高温库1巷道出库**)
	(*************************
	上位机通讯程序
	出口状态  D3105
	1:禁止出库
    2:允许出库
    收到空框请求D2105
    1：复位，
    2：收到出库请求
	**********************出库********************************)
	(******1巷道******)
	IF NOT XED AND Export1LoadCylinderIO.iDestinationPos=2 THEN
		D3105:=2;
	ELSE
		D3105:=1;
	END_IF;
	IF D2105=2 THEN
		M883:=1;
	ELSE
		M883:=0;
	END_IF;
	(******2巷道******)
   (*************************
	上位机通讯程序
	出口状态  D3125
	1:禁止出库
    2:允许出库
    收到空框请求D2115
    1：复位，
    2：收到出库请求
	**********************出库********************************)
	IF NOT XFD AND Export2LoadCylinderIO.iDestinationPos=2 THEN
		D3125:=2;
	ELSE
		D3125:=1;
	END_IF;
	IF D2120=2 THEN
		M884:=1;
	ELSE
		M884:=0;
	END_IF;
	(*********************入库****************************)
	(***********************************
	入口状态 D3100
	1:无电池入库请求
     2:有电池入库请求
	************************************)
	(******1巷道******)
	IF XE5 AND Import1LoadCylinderIO.iDestinationPos=2 THEN
		D3100:=2;
	ELSE
		D3100:=1;
    END_IF;  
    (******2巷道******)
    IF XF5 AND Import2LoadCylinderIO.iDestinationPos=2 THEN
		D3120:=2;
	ELSE
		D3120:=1;
    END_IF;
    (*******************************************************)
    (******高温出库分流******)
    (***********************************
	有板状态 D3305
	1：无板，2：有板
    分流方向 D2305
0：复位
1：读码失败
2：满筐进加压化成
3：满筐进二封
4：空筐回流进注液
	************************************)
	IF H3000SwitchPackageConveyorIn.xEmpty=0 THEN
		D3305:=1;
	ELSE
		D3305:=0;
	END_IF;
	IF D2305=2 THEN
		M882:=1;
	ELSE
		M882:=0;
	END_IF;
	(**********************************)
	 (******高温出库后升降机2分流******)
	     (***********************************
	有板状态 D3310
	1：无板，2：有板
    分流方向 D2310
0：复位
1：读码失败
2：空筐去注液
3：满筐去加压化成
	************************************)
	IF  Lifter2IO.iCurrentPos=5 AND Conveyor2IO.xEmpty=0 THEN
		D3310:=2;
	ELSE
		D3310:=1;
	END_IF;
	IF D2310=2 THEN
        Lifter2ExportChem:=0;
	END_IF;
	IF D2310=3 THEN
        Lifter2ExportChem:=1;
	END_IF;
	(***********************************)
	 
	IF  LDP(TRUE,M883) AND XED THEN
        Export1LoadCylinderIO.xMDIExe:=1;
        Export1LoadCylinderIO.iDestinationPos:=1;
	END_IF;
	IF NOT XED AND NOT Export1Conveyor1IO.xEmpty THEN
        Export1LoadCylinderIO.xMDIExe:=1;
        Export1LoadCylinderIO.iDestinationPos:=2;
     END_IF;		
	Export1Conveyor2IO.xLoad:=XED AND Export1LoadCylinderIO.iCurrentPos=1;
	Export1Conveyor2IO.xUnload:=Export1Conveyor1IO.xEmpty;
	Export1Conveyor1IO.xLoad:=Export1Conveyor2IO.xNextRun;
	IF Y1E5 THEN(*顶升移载前的挡停气缸，当挡停气缸有信号的时候要把1巷道的顶升移载落下*)
		Export1SwitchIO.xLiftCylinderExtendInit:=0;
	ELSE
		Export1SwitchIO.xLiftCylinderExtendInit:=1;
	END_IF;
	Export1Conveyor1Io.xUnload:=Export1SwitchConveyorIn.xEmpty;
	Export1SwitchIO.xEntryEnable:=Export1Conveyor1Io.xNextRun;
	Export1SwitchIO.xSwithEnable:=1;
	(*倍速链上只有一个物料出库*)
	Export1SwitchConveyorOut.xUnload:=H3000SwitchChemConveyorIn.xEmpty AND H3000SwitchPackageConveyorIn.xEmpty;
	(**高温库2巷道出库**)
	IF  LDP(TRUE,M884) AND XFD THEN
        Export2LoadCylinderIO.xMDIExe:=1;
        Export2LoadCylinderIO.iDestinationPos:=1;
	END_IF;
	IF NOT XFD AND NOT Export2Conveyor1IO.xEmpty THEN
        Export2LoadCylinderIO.xMDIExe:=1;
        Export2LoadCylinderIO.iDestinationPos:=2;
     END_IF;	
	Export2Conveyor1IO.xLoad:=XFD AND Export2LoadCylinderIO.iCurrentPos=1;
	Export2Conveyor1IO.xUnload:=Export2Conveyor2IO.xEmpty;
	Export2Conveyor2IO.xLoad:=Export2Conveyor1IO.xNextRun;
	Export2Conveyor2Io.xUnload:=Export2SwitchConveyorIn.xEmpty;
	Export2SwitchIO.xEntryEnable:=Export2Conveyor2Io.xNextRun;
	Export2SwitchIO.xSwithEnable:=1;
	Export2SwitchIO.xExitEnable:= NOT XE8; (*1巷道出库阻挡器检测*)
	IF Export1SwitchConveyorOut.xEmpty 
		AND Export1SwitchConveyorIn.xEmpty 
		AND Export1Conveyor1IO.xEmpty 
		AND XE8 THEN (*1巷道出库阻挡器检测*)
		Y1E5:=1;(*1巷道出库阻挡器*)
	ELSE
		Y1E5:=0;(*1巷道出库阻挡器*)

	END_IF;
	(*满框出库去二次封装线体*)
	H3000SwitchQuadPackageIO.xEntryEnable:=1;
	H3000SwitchQuadPackageIO.xSwithEnable:= NOT M882;(*触摸屏上按钮选择去化成还是去二封，后期通过上位机扫码给出*)
	IF H3000SwitchQuadPackageIO.xSwithEnable THEN
		H3000SwitchQuadPackageio.xExitEnable:=H3000Conveyor1IO.xEmpty;
		H3000Conveyor1Io.xLoad:=H3000SwitchPackageConveyorOut.xNextRun;
	ELSE
		H3000SwitchQuadPackageio.xExitEnable:=0;	
		H3000Conveyor1Io.xLoad:=0;
	END_IF;
	H3000Conveyor1IO.xUnload:=H3000Conveyor2IO.xEmpty;
	H3000Conveyor2IO.xLoad:=H3000Conveyor1IO.xNextRun;
	H3000Conveyor2IO.xUnload:=H3000Conveyor3IO.xEmpty;
	H3000Conveyor3IO.xLoad:=H3000Conveyor2IO.xNextRun;	
	H3000Conveyor3IO.xUnload:=H3000Conveyor4IO.xEmpty;
	H3000Conveyor4IO.xLoad:=H3000Conveyor3IO.xNextRun;
	H3000Conveyor4IO.xUnload:=H3000Conveyor5IO.xEmpty;
	H3000Conveyor5IO.xLoad:=H3000Conveyor4IO.xNextRun;
	H3000Conveyor5IO.xUnload:=H3000Conveyor6IO.xEmpty;
	H3000Conveyor6IO.xLoad:=H3000Conveyor5IO.xNextRun;
	H3000Conveyor6IO.xUnload:=H3000Conveyor7IO.xEmpty;
	H3000Conveyor7IO.xLoad:=H3000Conveyor6IO.xNextRun;
	H3000Conveyor7IO.xUnload:=H3000Conveyor8IO.xEmpty;
	H3000Conveyor8IO.xLoad:=H3000Conveyor7IO.xNextRun;	
	H3000Conveyor8IO.xUnload:=H3000Conveyor9IO.xEmpty;
	H3000Conveyor9IO.xLoad:=H3000Conveyor8IO.xNextRun;	
	H3000Conveyor9IO.xUnload:=H3000Conveyor10IO.xEmpty;
	H3000Conveyor10IO.xLoad:=H3000Conveyor9IO.xNextRun;
	H3000Conveyor10IO.xUnload:=D401.0;
	D201.0:=H3000Conveyor10IO.xNextRun;
    (**满框去化成**)
	H3000SwitchChemIO.xEntryEnable:=1;
	H3000SwitchChemIO.xSwithEnable:=1;
	H3000SwitchChemIO.xExitEnable:=H3000ChemConveyor2IO.xEmpty;
	H3000SwitchPackageConveyorIn.xUnload:=H3000SwitchChemConveyorIn.xEmpty;
	H3000ChemConveyor2IO.xLoad:=H3000SwitchChemConveyorOut.xNextRun;
	H3000ChemConveyor2IO.xUnload:=H3000ChemConveyor3IO.xEmpty;
	H3000ChemConveyor3IO.xLoad:=H3000ChemConveyor2IO.xNextRun;
	(*临时程序，Lifter2ExportChem:=1;以后要考虑空框回注液的程序，上位机扫码后判断是满框去化成还是空框去注液*)
	IF H3000ChemConveyor3IO.xEmpty=0 AND ( Lifter2TaskID=3 OR Lifter2TaskID=4)  THEN
		Lifter2IO.xMDIExe:=1;
		Lifter2IO.iDestinationPos:=5;
	END_IF;
	IF Lifter2IO.iCurrentPos=5 AND abs(D190-Lifter2Position[Lifter2IO.iDestinationPos])<10  THEN	
        Conveyor2IO.xLoad:=H3000ChemConveyor3IO.xNextRun;
        H3000ChemConveyor3IO.xUnload:=Conveyor2IO.xEmpty;
         Conveyor2IO.xloadCCW:=0;
	ELSE
		H3000ChemConveyor3IO.xUnload:=0;
	END_IF; 
	   IF Conveyor2IO.xEmpty=0 AND Lifter2TaskID=3 THEN
	   		Lifter2IO.xMDIExe:=1;
			Lifter2IO.iDestinationPos:=4;
	   END_IF;
	   	   IF Conveyor2IO.xEmpty=0 AND Lifter2TaskID=4 THEN
	   		Lifter2IO.xMDIExe:=1;
			Lifter2IO.iDestinationPos:=3;
	   END_IF;
	 IF Lifter2IO.iCurrentPos=4 AND abs(D190-Lifter2Position[Lifter2IO.iDestinationPos])<12  THEN	
	 	H2200Conveyor1IO.xLoad:=Conveyor2IO.xNextRun; 
	 	Conveyor2IO.xUnload:=H2200Conveyor1IO.xEmpty;
	 	Conveyor2IO.xUnloadCCW:=0;
	 END_IF;  
	      
	H2200Conveyor1IO.xUnload:=H2200Conveyor2IO.xEmpty;
	H2200Conveyor2IO.xLoad:=H2200Conveyor1IO.xNextRun;
	H2200Conveyor2IO.xUnload:=H2200Conveyor3IO.xEmpty;
	H2200Conveyor3IO.xLoad:=H2200Conveyor2IO.xNextRun;	
	H2200Conveyor3IO.xUnload:=H2200Conveyor4IO.xEmpty;
	H2200Conveyor4IO.xLoad:=H2200Conveyor3IO.xNextRun;
	H2200Conveyor4IO.xUnload:=H2200Conveyor5IO.xEmpty;
	H2200Conveyor5IO.xLoad:=H2200Conveyor4IO.xNextRun;
	H2200Conveyor5IO.xUnload:=H2200Conveyor6IO.xEmpty;
	H2200Conveyor6IO.xLoad:=H2200Conveyor5IO.xNextRun;
	H2200Conveyor6IO.xUnload:=H2200Conveyor7IO.xEmpty;
	H2200Conveyor7IO.xLoad:=H2200Conveyor6IO.xNextRun;
	H2200Conveyor7IO.xUnload:=H2200Conveyor8IO.xEmpty;
	H2200Conveyor8IO.xLoad:=H2200Conveyor7IO.xNextRun;	
	H2200Conveyor8IO.xUnload:=H2200Conveyor9IO.xEmpty;
	H2200Conveyor9IO.xLoad:=H2200Conveyor8IO.xNextRun;	
	H2200Conveyor9IO.xUnload:=H2200Conveyor10IO.xEmpty;
	H2200Conveyor10IO.xLoad:=H2200Conveyor9IO.xNextRun;
	H2200Conveyor10IO.xUnload:=D401.1;
	D201.1:=H2200Conveyor10IO.xNextRun;
	(*化成回流线体*)
	D201.2:=H1000Conveyor10IO.xEmpty;
	H1000Conveyor10IO.xLoad:=D401.2;
	H1000Conveyor10IO.xUnload:=H1000Conveyor9IO.xEmpty;
    H1000Conveyor9IO.xLoad:=H1000Conveyor10IO.xNextRun;
    H1000Conveyor9IO.xUnload:=H1000Conveyor8IO.xEmpty;
    H1000Conveyor8IO.xLoad:=H1000Conveyor9IO.xNextRun;
    H1000Conveyor8IO.xUnload:=H1000Conveyor7IO.xEmpty;
    H1000Conveyor7IO.xLoad:=H1000Conveyor8IO.xNextRun;
    H1000Conveyor7IO.xUnload:=H1000Conveyor6IO.xEmpty;
    H1000Conveyor6IO.xLoad:=H1000Conveyor7IO.xNextRun;
    H1000Conveyor6IO.xUnload:=H1000Conveyor5IO.xEmpty;
    H1000Conveyor5IO.xLoad:=H1000Conveyor6IO.xNextRun;
    H1000Conveyor5IO.xUnload:=H1000Conveyor4IO.xEmpty;
    H1000Conveyor4IO.xLoad:=H1000Conveyor5IO.xNextRun;
    H1000Conveyor4IO.xUnload:=H1000Conveyor3IO.xEmpty;
    H1000Conveyor3IO.xLoad:=H1000Conveyor4IO.xNextRun;
    H1000Conveyor3IO.xUnload:=H1000Conveyor2IO.xEmpty;
    H1000Conveyor2IO.xLoad:=H1000Conveyor3IO.xNextRun;  
    H1000Conveyor2IO.xUnload:=H1000Conveyor1IO.xEmpty;
    H1000Conveyor1IO.xLoad:=H1000Conveyor2IO.xNextRun; 
    IF H1000Conveyor1IO.xEmpty=0 AND Lifter2TaskID=2 THEN
    	Lifter2IO.xMDIExe:=1;
    	Lifter2IO.iDestinationPos:=2;
    END_IF;    
    IF Lifter2IO.iCurrentPos=2 AND abs(D190-Lifter2Position[Lifter2IO.iDestinationPos])<10  THEN 
    	H1000Conveyor1IO.xUnload:=Conveyor2IO.xEmpty;
     	Conveyor2IO.xLoad:=H1000Conveyor1IO.xNextRun;     	
    	Conveyor2IO.xloadCCW:=1;
    ELSE
    	H1000Conveyor1IO.xUnload:=0;
    END_IF;
   
	(*注液设备满框入库*)
	H850Conveyor4IO.xLoad:=M880;
	H850Conveyor4IO.xUnload:=H850Conveyor5IO.xEmpty;
	H850Conveyor5IO.xLoad:=H850Conveyor4IO.xNextRun;
	H850Conveyor5IO.xUnload:=H850Conveyor6IO.xEmpty;
	H850Conveyor6IO.xLoad:=H850Conveyor5IO.xNextRun;	
	IF H850RotorConveyorIO.xEmpty THEN
		 H850RotorIO.xMDIExe:=1;
		  H850RotorIO.iDestinationPos:=1;
	END_IF;
	IF H850RotorConveyorIO.xEmpty=0 THEN
		 H850RotorIO.xMDIExe:=1;
		  H850RotorIO.iDestinationPos:=2;
	END_IF;	
	IF H850RotorIO.iCurrentPos=1 THEN
    H850Conveyor6IO.xUnload:=H850RotorConveyorIO.xEmpty;
	ELSE
	 H850Conveyor6IO.xUnload:=0;
	END_IF;	
	H850RotorConveyorIO.xLoad:=H850Conveyor6IO.xNextRun;
	IF H850RotorIO.iCurrentPos=2 THEN
		H850RotorConveyorIO.xUnload:=H850SwitchConveyorIn.xEmpty AND H850SwitchConveyorOut.xEmpty;
	ELSE
		H850RotorConveyorIO.xUnload:=0;
	END_IF;
	H850SwitchIO.xEntryEnable:=H850RotorConveyorIO.xNextRun;	
	H850SwitchIO.xSwithEnable:=1;
	H850SwitchIO.xExitEnable:=H850Conveyor8IO.xEmpty;
    H850Conveyor8IO.xLoad:=H850SwitchConveyorOut.xNextRun;
    
    IF H850Conveyor8IO.xEmpty=0 AND Lifter2TaskID=1 THEN
    	Lifter2IO.xMDIExe:=1;
    	Lifter2IO.iDestinationPos:=1;
    END_IF;
    IF Lifter2IO.iCurrentPos=1 AND ABS(D190-Lifter2Position[Lifter2IO.iDestinationPos])<10 THEN
    	H850Conveyor8IO.xUnload:= Conveyor2IO.xEmpty;
    	Conveyor2IO.xLoad:=H850Conveyor8IO.xNextRun;
        Conveyor2IO.xloadCCW:=0;
    ELSE
    	H850Conveyor8IO.xUnload:=0;
    END_IF;
     IF (Lifter2TaskID=1 OR Lifter2TaskID=2 OR Lifter2TaskID=4) AND Conveyor2IO.xEmpty=0 THEN(*只要不是加压化成的 满框都要入库*)
     	Lifter2IO.xMDIExe:=1;
    	Lifter2IO.iDestinationPos:=3;
     END_IF;
    IF Lifter2IO.iCurrentPos=3 AND ABS(D190-Lifter2Position[Lifter2IO.iDestinationPos])<10 THEN	
		Conveyor2IO.xUnload:=H2200ImportConveyor2IO.xEmpty;
		H2200ImportConveyor2IO.xLoad:=Conveyor2IO.xNextRun;  
		Conveyor2IO.xUnloadCCW:=1;  	
    END_IF;
    (*不在目标位置不可下料*)
    IF ABS(D190-Lifter2Position[Lifter2IO.iDestinationPos])>12 THEN
    	Conveyor2IO.xUnload:=0;
    END_IF;
    IF H2200Switch1TaskID=5 THEN
	    H2200ImportConveyor2IO.xUnload:=H2200Switch1ConveyorOut.xEmpty;
	    H2200Switch1ConveyorOut.xLoad:=H2200ImportConveyor2IO.xNextRun;   
	    H2200Switch1IO.xLiftCylinderExtendInit:=1;	    
	    H2200Switch1ConveyorOut.xUnload:=H2200ImportConveyor1IO.xEmpty;   	    
    ELSE
    	 H2200ImportConveyor2IO.xUnload:=0;
    END_IF;
    H2200ImportConveyor1IO.xLoad:=H2200Switch1ConveyorOut.xNextRun;
    H2200ImportConveyor1IO.xUnload:=H2200Switch2ConveyorIn.xEmpty;
    H2200Switch2IO.xEntryEnable:=H2200ImportConveyor1IO.xNextRun;
    H2200Switch2IO.xSwithEnable:=1;
    H2200Switch2IO.xExitEnable:= Import1SwitchConveyorIn.xEmpty;(*此处有挡停后要加挡停条件，还要把巷道2的为空的条件加上*)
    (*1巷道入库*)
    Import1SwitchIO.xEntryEnable:=1;
    Import1SwitchIO.xSwithEnable:=1;
    Import1SwitchIO.xExitEnable:=Import1Conveyor1IO.xEmpty;
    Import1Conveyor1IO.xLoad:=Import1SwitchConveyorOut.xNextRun;
    Import1Conveyor1IO.xUnload:=Import1Conveyor2IO.xEmpty AND NOT XE5;
    Import1Conveyor2IO.xLoad:=Import1Conveyor1IO.xNextRun;
    
    IF Import1Conveyor2IO.xEmpty=0 AND XE5 THEN
    	Import1LoadCylinderIO.xMDIExe:=1;
    	Import1LoadCylinderIO.iDestinationPos:=2;
    	Import1Conveyor2IO.xPutInto:=0;
    END_IF;
    IF NOT XE5 THEN
    	Import1LoadCylinderIO.xMDIExe:=1;
    	Import1LoadCylinderIO.iDestinationPos:=1;	
    END_IF;
    IF LDP(TRUE, Import1LoadCylinderIO.iCurrentPos=1) THEN
    	Import1Conveyor2IO.xPutInto:=1;
    END_IF;
 (*2巷道入库*)
 
    Y173:=1;(*空框A返回倍速链*)
   Y175:=1;(*空框B返回倍速链*)
   (*空框回流*)
   H2200SwitchEmptyABackIO.xEntryEnable:=1;
   H2200SwitchEmptyABackIO.xLiftCylinderExtendInit:=1;
    H2200SwitchEmptyABackIO.xSwithEnable:=1;
    IF H2200Switch1TaskID=3  THEN
    	H2200SwitchEmptyABackIO.xExitEnable:=H2200Switch1ConveyorIn.xEmpty;   	
    	H2200Switch1IO.xEntryEnable:=H2200SwitchEmptyABackConveyorOut.xNextRun;
    	H2200Switch1IO.xSwithEnable:=0;
    	H2200Switch1IO.xExitEnable:=H2200RotorConveyorIO.xEmpty AND H2200RotorIO.iCurrentPos=1 AND X6F;
    ELSE
    	H2200SwitchEmptyABackIO.xExitEnable:=0;
    END_IF;
    IF H2200Switch1TaskID<>5 THEN
    	H2200Switch1IO.xLiftCylinderExtendInit:=0;
    END_IF;
    IF H2200RotorConveyorIO.xEmpty THEN
    	H2200RotorIO.xMDIExe:=1;
    	H2200RotorIO.iDestinationPos:=1;
    END_IF;
    IF H2200RotorConveyorIO.xEmpty=0 THEN
     	H2200RotorIO.xMDIExe:=1;
    	H2200RotorIO.iDestinationPos:=2;   
    END_IF;   
    IF H2200RotorIO.iCurrentPos=1 AND X6F THEN
    	H2200RotorConveyorIO.xLoad:=H2200Switch1ConveyorIn.xNextRun;
    ELSE
    	H2200RotorConveyorIO.xLoad:=0;	
    END_IF;
    IF Conveyor1IO.xEmpty THEN
    	Lifter1IO.xMDIExe:=1;
    	Lifter1IO.iDestinationPos:=2;
    END_IF;
    IF Conveyor1IO.xEmpty=0 THEN
    	Lifter1IO.xMDIExe:=1;
    	Lifter1IO.iDestinationPos:=1; 
    END_IF;
    IF Lifter1IO.iCurrentPos=2 AND X8D AND H2200RotorIO.iCurrentPos=2 AND X75 THEN
    	H2200RotorConveyorIO.xUnload:=Conveyor1IO.xEmpty;
    ELSE
    	H2200RotorConveyorIO.xUnload:=0;
    END_IF;
    Conveyor1IO.xLoad:=H2200RotorConveyorIO.xNextRun; 
    IF Lifter1IO.iCurrentPos=1 AND X8C THEN
    	Conveyor1IO.xUnload:=H850Conveyor3IO.xEmpty;
    ELSE
    	Conveyor1IO.xUnload:=0;
    END_IF;  	
    H850Conveyor3IO.xLoad:=Conveyor1IO.xNextRun;
    h850conveyor3IO.xUnload:=H850Conveyor1IO.xEmpty;
    H850Conveyor1IO.xLoad:=H850Conveyor3IO.xNextRun;
END_IF;

IF g_xManual THEN
    D201:=0;(*发送给化成B柜*)
    (************发送给上位机程序复位**************)
    D3016:=0;
    D3011:=0;
    (*****************************************************)
	IF M134 THEN (*空框A返回倍速链 手动*)
		 Y173:=1;(*空框A返回倍速链*)
	ELSE
		Y173:=0;;(*空框A返回倍速链*)
	END_IF;
	IF M135 THEN (*空框B返回倍速链 手动*)
		 Y175:=1;(*空框B返回倍速链*)
	ELSE
		Y175:=0;(*空框B返回倍速链*)
	END_IF;	
	IF M163 THEN (*入库倍速链 手动*)
		 Y186:=1;(*入库倍速链*)
	ELSE
		Y186:=0;;(*入库倍速链*)
	END_IF;
	IF M64 THEN (*出库倍速链 手动*)
		 Y187:=1;(*出库倍速链 *)
	ELSE
		Y187:=0;(*出库倍速链 *)
	END_IF;		
END_IF;
END_PROGRAM

PROGRAM Start
IF g_xReset THEN
	SM50:=1;
ELSE
	SM50:=0;
END_IF;
CASE g_iState OF
	0: 
		g_xManual:=1;
		g_xAuto:=0;	
		g_xStackLampAmber:=1;
		g_xStackLampGreen:=0;
		g_xRemoteAuto:=0;
	1:
		g_xManual:=0;
		g_xAuto:=1;
		g_xStackLampGreen:=1;
		g_xStackLampAmber:=0;
		g_xRemoteAuto:=0;
	2:	
        g_xRemoteAuto:=1;
        g_xStackLampGreen:=1;
        g_xStackLampAmber:=0;
        g_xAuto:=0;
		g_xManual:=0;
END_CASE;
IF g_xLocalAutoStart THEN  
	g_iState:=1;
END_IF;
IF g_xAlarm AND SM412 THEN
	g_xStackLampRed:=1;
	g_xBuzzer:=1;
ELSE
	g_xStackLampRed:=0;
	g_xBuzzer:=0;	
END_IF;
IF g_xStop OR g_xEStop=0 THEN 
	g_iState:=0;
END_IF;
IF g_xRemoteAutoStart THEN
	g_iState:=2;
END_IF;
END_PROGRAM

PROGRAM UDP
(*与化成柜2通讯*)
D200:=2;
SP_SOCOPEN( SM403 AND NOT SD1282.0 AND NOT SD1284.0 AND SD1288.A , "U0", K1 , D110 , M100);
SP_SOCSND( SM413 AND SD1282.0 , "U0" , K1 , D100, D200, M102 );
SP_SOCRCV( SD1282.0 AND SD1286.0 AND NOT M104 , "U0" , K1, D300 , D400 ,M104 );
SP_SOCCLOSE( LDF(TRUE,SD1082.0) , "U0" , K1, D120, M106 );
(*编码器处理程序*)
IF XA OR X0B   THEN
	D140:=2;
	D143:=6;
END_IF;
	G_INPUT( X0A OR X0B, 0 , D140 , D160 , M110 );(*串口数据读取指令*)
IF M110 THEN
	D170:=0;
	D172:=4;
END_IF;
ZP_CSET( M110  , "U0", 2 , D170, D180,M112 );(*串口数据缓存区清除指令*)
IF D160=11069 THEN  (*接收到数据开始执行ASCII码转换成10进制，D160为=+ ，串口传输的字头 转换为10进制是11069，不判断这个报4100错误*)
    DABIN( TRUE , D163, D190 );
END_IF;
END_PROGRAM

FUNCTION_BLOCK Conveyor
VAR
  m_tLoadTimer : TIME;  (* 上料延时 *)
  m_tonNotArriveAlarm : TON;  (* 未到达报警计时 *)
  m_tonUnloadAlam : TON;  (* 下料报警定时器 *)
  m_tonLoadDelay : TON;  (* 上料延时 *)
  m_tUnloadTimer : TIME;  (* 下料计时器 *)
  iStep : INT;  (* 上料步骤 *)
  m_tNotArriveCurrentTime : TIME;  (* 未到达报警计时当前时间 *)
  m_xInitial : BOOL;  (* 初始化 *)
  m_xLoadDelayOut : BOOL;  (* 上料延时输出 *)
END_VAR
VAR_IN_OUT
  ConveyorMotor : ConveyorIO;  (* 输送线输入输出 *)
END_VAR
(*////////////////////////////////////////////////////////////////////////////////////////////////////////////
//传输线控制FB块，可控制单方向线体，双向旋转线体，支持双向上下料            
//线体初始化后为空的情况下输入xLoad信号即可进行上料动作，使用xLoadCCW信号可反方向上料
//增加了产品信息和产品种类的储存，当传输线为空和上料进行标志位为零的情况下清除产品信息和产品种类
//使用方式是在置位xLoad信号后，把产品信息和产品种类传入，等下料后自动清零
//线体不为空的情况下使用xUnload信号可进行下料动作，物料有无传感器的下降沿后出发计时器，延时断开传输线旋转
//单方向传输线体把xLoadCCW、xUnloadCCW设置为零，双向线体上料方向和下料反向的,方向固定的 把xUnloadCCW设置为1
//双方向线体双向都能上下料的要根据上料的方向来设置xLoadCCW,xUnloadCCW
//增加工作中信号xBusy当电机正转 显示为工作中
//增加上下料超时报警，xLoadAlarm，xUnloadAlarm，设定时间在LOAD_UNLOAD_TIME常量上，现在设置的为30秒
//增加xPutInto信号，用于直接投入的物料，检测开关感应到后，直接进入下料流程，上升沿有效
//离开延时改为变量 iLeaveDelay 默认为0 离开检测开关离输送线尾端比较远的线体需要根据情况设定100ms为单位
增加初始化标志位，增加进入延时时间，初始化为进入延时时间为0 ，离开延时时间为2S，通过外围接口可以更改
//修改信息  修改后请增加版本
12-17进行了优化，增加了未到达报警，当物料未传送到下一设备，就报未到达报警，使用xNextRun标志位制作，没有正常到达
第0步，不能跳转到第一步把标志位复位，即出现中断情况，2秒后报警
//YAO      V1.0
///////////////////////////////////////////////////////////////////////////////////////////////////////////
********************************************************)
IF NOT m_xInitial THEN
	ConveyorMotor.tLoadDelay:=T#0s;
	ConveyorMotor.tUnloadAlarmDelay:=T#30s;
	m_xInitial:=1;
END_IF;

CASE iStep OF
	0:
	ConveyorMotor.xMotorCW:=0;
	ConveyorMotor.xMotorCCW:=0;
    IF g_xAuto THEN
		IF (ConveyorMotor.xCWPresent OR ConveyorMotor.xCCWPresent)  THEN
			iStep:=3;
			ConveyorMotor.xEmpty:=0;
			ELSE
			iStep:=1;
			ConveyorMotor.xEmpty:=1;
		END_IF;
	END_IF;
	1: 
	ConveyorMotor.xNextRun:=0;
	IF ConveyorMotor.xLoad AND ConveyorMotor.xEmpty THEN	
		iStep:=2;
	END_IF;
	2: 
	IF ConveyorMotor.xloadCCW THEN
		ConveyorMotor.xMotorCCW:=1; 
		ConveyorMotor.xMotorCW:=0;
	ELSE
	    ConveyorMotor.xMotorCW:=1;  
		ConveyorMotor.xMotorCCW:=0;
	END_IF;
		m_tonLoadDelay(IN:= (ConveyorMotor.xCWPresent AND NOT ConveyorMotor.xloadCCW) 
		                                        OR (ConveyorMotor.xCCWPresent AND ConveyorMotor.xloadCCW) ,
		                               PT:= ConveyorMotor.tLoadDelay ,
		                               Q:= m_xLoadDelayOut ,
		                               ET:= m_tLoadTimer );
	    IF m_xLoadDelayOut THEN 	 
		    iStep:=3;
		END_IF;
	3:
	ConveyorMotor.xMotorCW:=0;
	ConveyorMotor.xMotorCCW:=0;
	ConveyorMotor.xEmpty:=0;
	IF ConveyorMotor.xUnload THEN 
		iStep:=4;
	END_IF;
	4:	
	IF ConveyorMotor.xUnloadCCW THEN   
		ConveyorMotor.xMotorCCW:=1;  
		ConveyorMotor.xMotorCW:=0;
		ELSE
	    ConveyorMotor.xMotorCW:=1;  
		ConveyorMotor.xMotorCCW:=0;
	END_IF;
	ConveyorMotor.xNextRun:=1; 
	IF NOT ConveyorMotor.xUnload THEN 
		istep:=0;
	END_IF;
END_CASE;
IF LDP(TRUE,ConveyorMotor.xPutInto) THEN
	iStep:=0;
END_IF;

(*IF ConveyorMotor.xEmpty AND iStep<>2 THEN
	ConveyorMotor.iProductCategory:=0;
END_IF;*)
IF g_xEStop=0 OR g_xReset THEN
	iStep:=0;
END_IF;	
IF g_xReset THEN
	ConveyorMotor.xNextRun:=0; 
END_IF;
IF g_xManual THEN
	iStep:=0;
	IF ConveyorMotor.xForward 
		AND ConveyorMotor.xBackward=0 
		AND ConveyorMotor.xMotorCCW=0
		AND g_xEStop THEN
		ConveyorMotor.xMotorCW:=1;
		ConveyorMotor.xMotorCCW:=0;
		ELSE
		ConveyorMotor.xMotorCW:=0;
	END_IF;

	IF ConveyorMotor.xBackward 
		AND ConveyorMotor.xForward=0 
		AND ConveyorMotor.xMotorCW=0
		AND g_xEStop  THEN
		ConveyorMotor.xMotorCCW:=1;
		conveyormotor.xMotorCW:=0;
		ELSE
		ConveyorMotor.xMotorCCW:=0;
	END_IF;
END_IF;
IF ConveyorMotor.xMotorCCW        
	OR ConveyorMotor.xMotorCW THEN  
	ConveyorMotor.xBusy:=1;
	ELSE
	ConveyorMotor.xBusy:=0;
END_IF;
m_tonNotArriveAlarm(IN:= iStep=0 AND ConveyorMotor.xNextRun  ,PT:= T#2s,Q:= ConveyorMotor.xNotArriveAlarm ,ET:= m_tNotArriveCurrentTime );
m_tonUnloadAlam(IN:= iStep=4,PT:=ConveyorMotor.tUnloadAlarmDelay,Q:= ConveyorMotor.xUnloadAlarm,ET:= m_tUnloadTimer );
END_FUNCTION_BLOCK

FUNCTION_BLOCK ShuttleCar
VAR_IN_OUT
  ShuttleCarInOut : ShuttleCarIO;
END_VAR
VAR
  m_xBrakeDelay : BOOL;  (* 刹车延时标志位 *)
  diCurrentPosRetain : DINT;
  m_tonBrakeDelay : TON;  (* 延时 *)
  m_tBrakeDelay : TIME;
  m_xBrake : BOOL;
  m_tBrakeDelayCurrentTime : TIME;
END_VAR
(*******************************************************************
输送小车程序，可用于使用认址片控制位置的输送车程序，可用于控制提升机，
使用了限位捕捉程序防止小车惯性过大冲过限位后继续行走，捕捉程序采用反
转复位，这样设计有弊端可能反转复位后车的位置并没有回到限位以内,当两个
限位同时碰到的时候，会使运料小车进入死锁状态，通过xPassLimit来解开死锁，
可以在触摸屏中使用一个带权限的按钮来进行控制，配合ShuttleCarCurrentPos
函数来计算位置信息
增加自动开始后将当前位置置为零的信号防止设备停在两个位置开关的中间
修改信息  修改后请增加版本
YAO      V1.0
********************************************************************)

ShuttleCarInOut.xPosLimitCatch:=LDF(TRUE,ShuttleCarInOut.xPosLimit) OR ShuttleCarInOut.xPosLimitCatch;
IF ShuttleCarInOut.xCCW THEN  
	ShuttleCarInOut.xPosLimitCatch:=0;
END_IF;

ShuttleCarInOut.xNegLimitCatch:=LDF(TRUE,ShuttleCarInOut.xNegLimit) OR ShuttleCarInOut.xNegLimitCatch;
IF ShuttleCarInOut.xCW THEN   
	ShuttleCarInOut.xNegLimitCatch:=0;  
END_IF;
IF ShuttleCarInOut.xPassLimit OR
	(ShuttleCarInOut.xNegLimitCatch 
	AND ShuttleCarInOut.xPosLimitCatch)  THEN  
	ShuttleCarInOut.xNegLimitCatch:=0; 
	ShuttleCarInOut.xPosLimitCatch:=0;
END_IF;

IF ShuttleCarInOut.xReady THEN	
    IF g_xManual THEN  
	    IF ShuttleCarInOut.xForward 
			AND ShuttleCarInOut.xBackward=0 
			AND ShuttleCarInOut.xCCW=0 
			AND ShuttleCarInOut.xPosLimitCatch=0 
			AND g_xEStop THEN
		    ShuttleCarInOut.xCW:=1;
		    ELSE
		    ShuttleCarInOut.xCW:=0;
	    END_IF;
	    IF ShuttleCarInOut.xBackward 
			AND ShuttleCarInOut.xForward=0 
			AND ShuttleCarInOut.xCW=0 
			AND ShuttleCarInOut.xNegLimitCatch=0 
			AND G_xEStop THEN  
		    ShuttleCarInOut.xCCW:=1;
		    ELSE
		    ShuttleCarInOut.xCCW:=0;
	    END_IF;
    END_IF;
  IF g_xAuto AND g_xEStop THEN  
	  IF ShuttleCarInOut.xMDIExe AND ShuttleCarInOut.iDestinationPos<>0 THEN
	
	    IF ShuttleCarInOut.iCurrentPos<ShuttleCarInOut.iDestinationPos AND ShuttleCarInOut.xPosLimitCatch=0 THEN
			ShuttleCarInOut.xCW:=1;
			ShuttleCarInOut.xCCW:=0;
			ShuttleCarInOut.xMDIDone:=0;
		END_IF;

		IF ShuttleCarInOut.iCurrentPos>ShuttleCarInOut.iDestinationPos AND ShuttleCarInOut.xNegLimitCatch=0 THEN
			ShuttleCarInOut.xCCW:=1;
			ShuttleCarInOut.xCW:=0;
			ShuttleCarInOut.xMDIDone:=0;
		END_IF;
	
		IF ShuttleCarInOut.iCurrentPos=ShuttleCarInOut.iDestinationPos THEN
			ShuttleCarInOut.xCW:=0;
			ShuttleCarInOut.xCCW:=0;
			ShuttleCarInOut.xMDIDone:=1;
			ELSE
			ShuttleCarInOut.xMDIDone:=0;
		END_IF;

		IF ShuttleCarInOut.xPosLimitCatch THEN
			ShuttleCarInOut.xCW:=0;
			ShuttleCarInOut.xMDIDone:=0;
		END_IF;

		IF ShuttleCarInOut.xNegLimitCatch THEN
			ShuttleCarInOut.xCCW:=0;
			ShuttleCarInOut.xMDIDone:=0;
		END_IF;
		ELSE
		ShuttleCarInOut.xCW:=0;
		ShuttleCarInOut.xCCW:=0;
		ShuttleCarInOut.xMDIDone:=0;
	  END_IF;
	END_IF;
	ELSE
		ShuttleCarInOut.xCW:=0;
		ShuttleCarInOut.xCCW:=0;	
END_IF;
m_tonBrakeDelay(IN:=m_xBrakeDelay ,PT:= T#100ms,Q:=m_xBrake ,ET:= m_tBrakeDelayCurrentTime);
IF (ShuttleCarInOut.xCW OR ShuttleCarInOut.xCCW) AND ShuttleCarInOut.xReady=1 THEN
	ShuttleCarInOut.xBrake:=m_xBrake;
	m_xBrakeDelay:=1;
	ELSE
	ShuttleCarInOut.xBrake:=0;
	m_xBrakeDelay:=0;
END_IF;

IF g_xEStop =0 THEN
	ShuttleCarInOut.xCW :=0;
	ShuttleCarInOut.xCCW:=0;
END_IF;

(*IF SM402 THEN 
	ShuttleCarInOut.diCurrentPos:=diCurrentPosRetain;
	ELSE
	diCurrentPosRetain:=ShuttleCarInOut.diCurrentPos;
END_IF;*)
(*自动上电后把当前位置清零，防止穿梭车不在开关位置*)
IF LDP(TRUE,g_xAuto) THEN
	ShuttleCarInOut.iCurrentPos:=0;
END_IF;
IF ShuttleCarInOut.xCW OR ShuttleCarInOut.xCCW THEN
	ShuttleCarInOut.xBusy:=1;
	ELSE
	ShuttleCarInout.xBusy:=0;
END_IF;
END_FUNCTION_BLOCK

FUNCTION ShuttleCarCurrentPosition
VAR_INPUT
  xPosition1 : BOOL;
  xPosition2 : BOOL;
  xPosition3 : BOOL;
END_VAR
(************************************
计算输送车当前位置的函数
**************************************)
IF xPosition1 THEN
	ShuttleCarCurrentPosition:=1;
END_IF;
IF xPosition2 THEN
	ShuttleCarCurrentPosition:=2;
END_IF;
IF xPosition3 THEN
	ShuttleCarCurrentPosition:=3;
END_IF;
END_FUNCTION

FUNCTION_BLOCK Switch
VAR_IN_OUT
  ConveyorEntryIO : ConveyorIO;
END_VAR
VAR
  ConveyorEntry : Conveyor;
END_VAR
VAR_IN_OUT
  ConveyorExitIO : ConveyorIO;
END_VAR
VAR
  m_tonLiftCylinderDelay : TON;  (* 顶升延时 *)
  m_xLiftCylinderDelay : BOOL;
  m_tLiftCylinderDelay : TIME;
  m_tonExitBarDelay : TON;  (* 退出阻挡器延时 *)
  m_tExitBarDelay : TIME;
  m_xExitBarDelay : BOOL;
END_VAR
VAR_IN_OUT
  SwitchIO : SwitchIO;
END_VAR
VAR
  iStep : INT;
  ConveyorExit : Conveyor;
  m_xInitial : BOOL;
END_VAR
(**************************************************
顶升移载模块，抽象为一条输入输送线 ，一条输出输送线
一个进入阻挡器，一个放出阻挡器，和一个顶升气缸的控制
程序思路比较混乱，接口不清晰，需要整改
12-17日   V1.0
***************************************************)
ConveyorEntry(ConveyorMotor:=ConveyorEntryIO);
ConveyorExit(ConveyorMotor:=ConveyorExitIO);

IF NOT m_xInitial THEN
	
	m_xInitial:=1;
END_IF;
IF g_xAuto THEN
	CASE iStep OF
		0:(*初始化*)
		ConveyorEntryIO.xLoad:=0;
		ConveyorEntryIO.xUnload:=0;
		ConveyorEntryIO.xPutInto:=0;
		ConveyorExitIO.xLoad:=0;
		ConveyorExitIo.xUnload:=0;
		ConveyorExitIO.xPutInto:=0;
		SwitchIO.xEntryBarCylinderRetract:=0;
		SwitchIO.xExitBarCylinderRetract:=0;
		IF SwitchIO.xLiftCylinderExtendInit THEN
			SwitchIO.xLiftCylinderExtend:=1;
			SwitchIO.xLiftCylinderRetract:=0;
		    IF SwitchIO.xLiftCylinderExtendDetect THEN
			    iStep:=1;
		     END_IF; 
		ELSE
			SwitchIO.xLiftCylinderExtend:=0;
			SwitchIO.xLiftCylinderRetract:=1;	
		    IF SwitchIO.xLiftCylinderRetractDetect THEN
			    iStep:=1;
		    END_IF;		
		END_IF;
		1:(*上料*)
        IF SwitchIO.xEntryEnable AND ConveyorEntryIO.xEmpty AND ConveyorExitIO.xEmpty THEN
        	SwitchIO.xEntryBarCylinderRetract:=1;
        	ConveyorEntryIO.xLoad:=1;
        END_IF;
        IF ConveyorEntryIO.xEmpty=0 THEN
        	SwitchIO.xEntryBarCylinderRetract:=0;
        	ConveyorEntryIO.xLoad:=0;
        	ConveyorExitIO.xPutInto:=1;
        END_IF;
        IF m_xLiftCylinderDelay AND  SwitchIO.xSwithEnable THEN
        	 iStep:=2;
        END_IF;
        IF SwitchIO.xSwithEnable=0 AND m_xLiftCylinderDelay  THEN
        	 iStep:=3;
        END_IF;
		2:(*顶升*)
			SwitchIO.xExitBarCylinderRetract:=0;
		    IF SwitchIO.xLiftCylinderExtendInit THEN
			    SwitchIO.xLiftCylinderExtend:=0;
			    SwitchIO.xLiftCylinderRetract:=1;
		    ELSE
			    SwitchIO.xLiftCylinderExtend:=1;
			    SwitchIO.xLiftCylinderRetract:=0;			
		   END_IF;

		  IF SwitchIO.xLiftCylinderExtendInit THEN
		  	IF SwitchIO.xLiftCylinderRetractDetect THEN
		  		iStep:=4;
		  	END_IF;
		  	ELSE
		  	IF SwitchIO.xLiftCylinderExtendDetect THEN
		      iStep:=4; 
		  	END_IF;
		  END_IF;
		  3:(*放行*)	
		  	SwitchIO.xExitBarCylinderRetract:=1;
		  	iStep:=4;
		  4:(*下料*)
		  (*通过出料传输线下料*)
		  IF SwitchIO.xExitEnable  AND m_xExitBarDelay AND NOT SwitchIO.xExitBarCylinderRetract  THEN		  
		  	ConveyorExitIO.xUnload:=1;
		  ELSE
		  	ConveyorExitIO.xUnload:=0;
		  END_IF;	
		   (*通过进料传输线下料*)
		  IF SwitchIO.xExitEnable  AND m_xExitBarDelay  AND SwitchIO.xExitBarCylinderRetract THEN		  
		  	ConveyorEntryIO.xUnload:=1;
		  ELSE
		  	ConveyorEntryIO.xUnload:=0;
		  END_IF;			    	
		  IF ConveyorExitIO.xEmpty OR ConveyorEntryIO.xEmpty  THEN
		  	ConveyorExitIO.xPutInto:=1;
		  	ConveyorEntryIO.xPutInto:=1;
			iStep:=0; 
		  END_IF;
	END_CASE;
        m_tonLiftCylinderDelay(IN:=NOT ConveyorEntryIO.xEmpty AND iStep=1 ,PT:= T#1S ,Q:= m_xLiftCylinderDelay ,ET:=m_tLiftCylinderDelay );
 		m_tonExitBarDelay(IN:=iStep=4 ,PT:= T#1s ,Q:= m_xExitBarDelay ,ET:= m_tExitBarDelay);
END_IF;
IF g_xReset OR LDP(TRUE,SwitchIO.xLiftCylinderExtendInit) OR LDF(TRUE,SwitchIO.xLiftCylinderExtendInit) THEN
	iStep:=0;
END_IF;
IF g_xManual  THEN
	iStep:=0;
	ConveyorEntryIO.xLoad:=0;
    ConveyorEntryIO.xUnload:=0;
	ConveyorEntryIO.xPutInto:=0;
	ConveyorExitIO.xLoad:=0;
	ConveyorExitIo.xUnload:=0;
	ConveyorExitIO.xPutInto:=0;
	SwitchIO.xEntryBarCylinderRetract:=0;
	SwitchIO.xExitBarCylinderRetract:=0;
	IF SwitchIO.xEntryBarCylinderRetractButton THEN
		SwitchIO.xEntryBarCylinderRetract:=1;
	ELSE
		SwitchIO.xEntryBarCylinderRetract:=0;
	END_IF;
		IF SwitchIO.xExitBarCylinderRetractButton THEN
		SwitchIO.xExitBarCylinderRetract:=1;
	ELSE
		SwitchIO.xExitBarCylinderRetract:=0;
		END_IF;
		IF SwitchIO.xLiftCylinderExtendButton AND NOT SwitchIO.xLiftCylinderRetractButton THEN
			SwitchIO.xLiftCylinderExtend:=1;
			SwitchIO.xLiftCylinderRetract:=0;
		END_IF;
		IF NOT SwitchIO.xLiftCylinderExtendButton AND  SwitchIO.xLiftCylinderRetractButton THEN
			SwitchIO.xLiftCylinderExtend:=0;
			SwitchIO.xLiftCylinderRetract:=1;
		END_IF;		
	END_IF;
END_FUNCTION_BLOCK

FUNCTION ShuttleCarVelocityEncoder
VAR_INPUT
  iDestinationPos : INT;  (* 目标位置 *)
  iCurrentPos : INT;  (* 当前位置 *)
  xEnable : BOOL;  (* 使能 *)
END_VAR
IF xEnable THEN
	IF ABS(iCurrentPos-iDestinationPos)<200  THEN
		ShuttleCarVelocityEncoder:=0;
	ELSE
		ShuttleCarVelocityEncoder:=1;
	END_IF;
ELSE
	ShuttleCarVelocityEncoder:=0;
END_IF;
END_FUNCTION

FUNCTION_BLOCK PriorityFB
VAR_INPUT
  xCondition1 : BOOL;  (* 条件1 *)
  xCondition2 : BOOL;  (* 条件2 *)
  xCondition3 : BOOL;  (* 条件3 *)
  xCondition4 : BOOL;  (* 条件4 *)
  xCondition5 : BOOL;  (* 条件5 *)
  xTaskComplete : BOOL;  (* 任务完成 *)
  xReset : BOOL;  (* 复位 *)
END_VAR
VAR
  xOccupy : BOOL;  (* 占用 *)
END_VAR
VAR_OUTPUT
  iPriority : INT;  (* 输出任务号 *)
END_VAR
IF xCondition1 AND NOT xOccupy THEN
	iPriority:=1;
	xOccupy:=1;
END_IF;
IF xCondition2 AND NOT xOccupy THEN
	iPriority:=2;
	xOccupy:=1;
END_IF;
IF xCondition3 AND NOT xOccupy THEN
	iPriority:=3;
	xOccupy:=1;
END_IF;
IF xCondition4 AND NOT xOccupy THEN
	iPriority:=4;
	xOccupy:=1;
END_IF;
IF xCondition5 AND NOT xOccupy THEN
	iPriority:=5;
	xOccupy:=1;
END_IF;
IF NOT xCondition1 
	AND NOT xCondition2
	AND NOT xCondition3
	AND NOT xCondition4
	AND NOT xCondition5
	AND NOT xOccupy  THEN
	iPriority:=0;
END_IF;
IF LDP(TRUE, xTaskComplete) THEN
	xOccupy:=0;
	iPriority:=0;
END_IF;
IF xReset THEN
	iPriority:=0;
END_IF;
END_FUNCTION_BLOCK

FUNCTION_BLOCK ShuttleCarVelocityFB
VAR_INPUT
  xEnable : BOOL;  (* 使能 *)
  xMotorCW : BOOL;  (* 电机正转 *)
  xMotorCCW : BOOL;  (* 电机反转 *)
  xPosition1Switch : BOOL;  (* 位置1开关 *)
  xDecelerationSwitch : BOOL;  (* 减速开关 *)
  xPosition2Switch : BOOL;  (* 位置2开关 *)
END_VAR
VAR
  iFloor : INT;  (* 层数 *)
END_VAR
VAR_OUTPUT
  xHighSpeed : BOOL;
END_VAR
IF xEnable THEN
	(*电机旋转，并且在位置开关上的时候触发加速*)
	IF( LDP(TRUE,xMotorCW) AND xPosition1Switch ) OR (  LDP(TRUE,xMotorCCW) AND xPosition2Switch) THEN
		xHighSpeed:=1;
		iFloor:=0;
	END_IF;
	IF LDF(TRUE,xMotorCW) OR LDF(TRUE,xMotorCCW) THEN
		xHighSpeed:=0;
    END_IF;
	IF LDP(TRUE,xDecelerationSwitch) THEN
		iFloor:=iFloor+1;
	END_IF;
	IF iFloor=2 THEN
		xHighSpeed:=0;
		iFloor:=0;
	END_IF;
ELSE
    xHighSpeed:=0;
END_IF;
END_FUNCTION_BLOCK
